(* Logix 5000 project; controller RN21_Architecture 1769-L16ER-BB1B rev 35.11; software revision 35.00; part 9 of 9 *)
(* tags used below, declared in another part *)
   Delformovingupdatedtimertonewpswd : TIMER;
   EmgLoginDn : BOOL;
   ExpDays_NoofattemptsLeft_visb : BOOL;
   ExpDays_NoofattemptsLeft_visbility : BOOL;
   ExpiryDays_MovFrmSrv : DINT;
   FC_RP_Arch : AOI_RP_Arch;
   FCI_PrintInterval : INT;
   FCI_RPDataLogTrig : BOOL;
   HMI_ChangePswd : BOOL;
   HMI_CONTROL_SCREEN : DINT;
   INTERNAL_RN21_HB_PLC2ServerCommFailed : BOOL;
   Lockout_Visb : BOOL;
   Logged_User : STRING;
   MaskTag : STRING;
   MaskTag1 : STRING;
   New_Pswd : STRING;
   New_Pswd_mask : STRING;
   New_Pswd_mask1 : STRING;
   Password_Change_Yes_Button_In_HMI : BOOL;
   PLC_RTC : DINT[7];
   Pswd_UpadatedSuccessfully : BOOL;
   pwdons : BOOL;
   RecipeEntryFloat : REAL[20];
   RecipeEntryInt : INT[11];
   RM_Param1 : DINT;
   RM_Param10 : REAL;
   RM_Param2 : DINT;
   RM_Param3 : DINT;
   RM_Param4 : DINT;
   RM_Param5 : DINT;
   RM_Param6 : REAL;
   RM_Param7 : REAL;
   RM_Param8 : REAL;
   RM_Param9 : REAL;
   RN21_BMAN_HMIBatchStart : BOOL;   // BATCH START
   RN21_LBStatus : INT;   // Login Block Status
   RN21_RM_LOADDLYBIT : BOOL;
   RN21_UM_ActiveUserMovFrmSrv : DINT;
   RN21_UM_Empty : STRING;   // Whenever Logout Will happen moving the Empty
   RN21_UM_ExpiryBitMovFrmSrv : DINT;
   RN21_UM_HMIPSWD_Visb : BOOL;
   RN21_UM_HMIPSWDAPPLY : BOOL;
   RN21_UM_HMIUserIDApply : BOOL;
   RN21_UM_HMIUSERPSWD : STRING;
   RN21_UM_INVALIDUserLatch : BOOL;
   RN21_UM_MaintBit : BOOL;
   RN21_UM_OperBit : BOOL;
   RN21_UM_Status_Visb : BOOL;
   RN21_UM_SupBit : BOOL;
   RN21_UM_USERIDEquLatch : BOOL;
   RN21_UM_USERIDMovFrmSrv : STRING;
   RN21_UM_UserLogout : BOOL;
   RN21_UM_UserLvlMovFrmSrv : DINT;
   RN21_UMAdmBit : BOOL;
   RN21_UMLogoutTag : INT;
   RN21_UMONS : DINT;
   RN21_UserLoginDN : BOOL;
   RP_Param1 : DINT;
   RP_Param10 : REAL;
   RP_Param2 : DINT;
   RP_Param3 : DINT;
   RP_Param4 : DINT;
   RP_Param5 : DINT;
   RP_Param6 : REAL;
   RP_Param7 : REAL;
   RP_Param8 : REAL;
   RP_Param9 : REAL;
   RPSrc : UDT_Recipe;
   RPSrc_RP_UID : DINT;
   TMR_LOGOUT : TIMER;
   TMR_UMLogoutTag : TIMER;
   TMR_UserIDRstDly : TIMER;
   TMRHMIPSWDVisb_Dly : TIMER;
   UM_Status1 : DINT;
   DummyBit : BOOL;
   EmergencyLoginActivated_Bit : BOOL;
   EmergencyUserIDEqual : BOOL;
   EmergencyUserPaswdEqual : BOOL;
   RN21_EmgUserID : STRING;
   RN21_UM_EmgPSWD : STRING;
   RP_Trigger : BOOL;
   RP_UID : DINT;
   RPSer : UDT_Recipe;
   UM_ACT : DINT;
   UM_Confirmation_Bit : BOOL;
   UM_EXPIRY : DINT;
   UM_EXPIRY_DAYS : DINT;
   UM_lockoutDurationLeft : DINT;
   UM_LVL : DINT;
   UM_NoOfAttempts : DINT;
   UM_PWD : STRING;
   UM_Status : DINT;
   UM_UID : STRING;
   UM_UID_OUT : STRING;
   UM_UniqueID : DINT;
(* MainProgram, continued *)

ROUTINE RN21_RM_Map   (* ladder *)
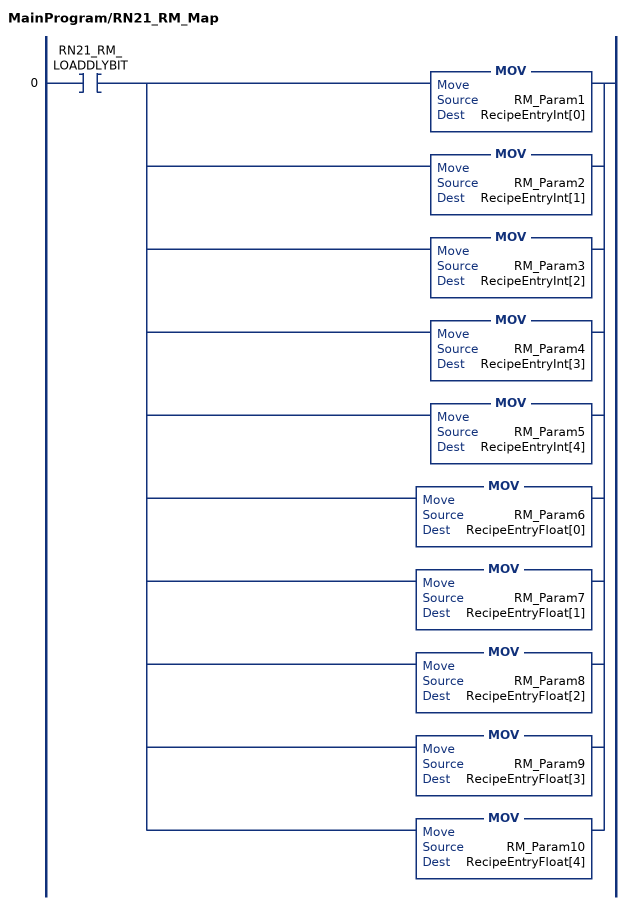
   0: XIC(RN21_RM_LOADDLYBIT)[MOV(RM_Param1,RecipeEntryInt[0]) ,MOV(RM_Param2,RecipeEntryInt[1]) ,MOV(RM_Param3,RecipeEntryInt[2]) ,MOV(RM_Param4,RecipeEntryInt[3]) ,MOV(RM_Param5,RecipeEntryInt[4]) ,MOV(RM_Param6,RecipeEntryFloat[0]) ,MOV(RM_Param7,RecipeEntryFloat[1]) ,MOV(RM_Param8,RecipeEntryFloat[2]) ,MOV(RM_Param9,RecipeEntryFloat[3]) ,MOV(RM_Param10,RecipeEntryFloat[4]) ];
END_ROUTINE

ROUTINE RN21_RP_Main   (* ladder *)
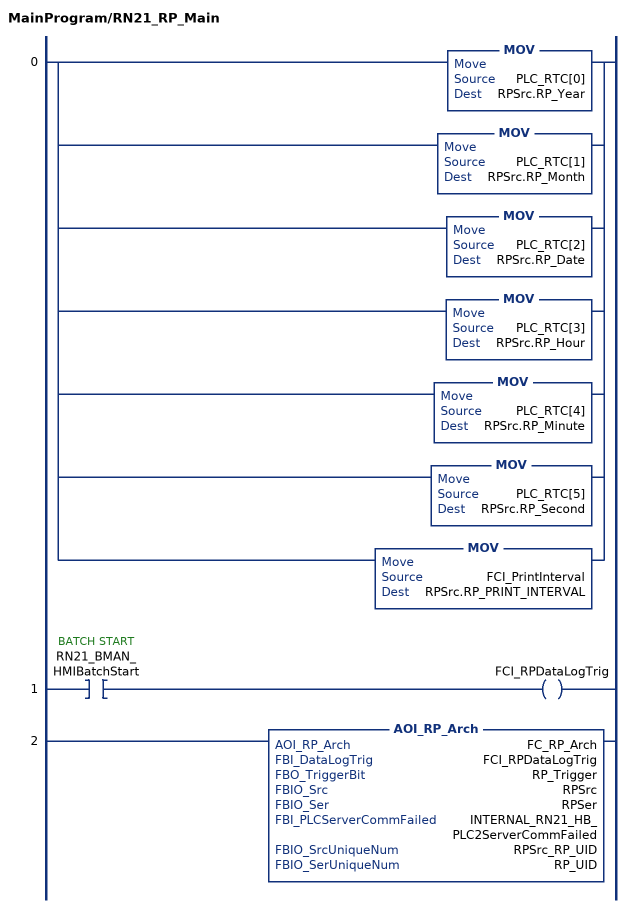
   0: [MOV(PLC_RTC[0],RPSrc.RP_Year) ,MOV(PLC_RTC[1],RPSrc.RP_Month) ,MOV(PLC_RTC[2],RPSrc.RP_Date) ,MOV(PLC_RTC[3],RPSrc.RP_Hour) ,MOV(PLC_RTC[4],RPSrc.RP_Minute) ,MOV(PLC_RTC[5],RPSrc.RP_Second) ,MOV(FCI_PrintInterval,RPSrc.RP_PRINT_INTERVAL) ];
   1: XIC(RN21_BMAN_HMIBatchStart)OTE(FCI_RPDataLogTrig);
   2: AOI_RP_Arch(FC_RP_Arch,FCI_RPDataLogTrig,RP_Trigger,RPSrc,RPSer,INTERNAL_RN21_HB_PLC2ServerCommFailed,RPSrc_RP_UID,RP_UID);
END_ROUTINE

ROUTINE RN21_RP_Map   (* ladder *)
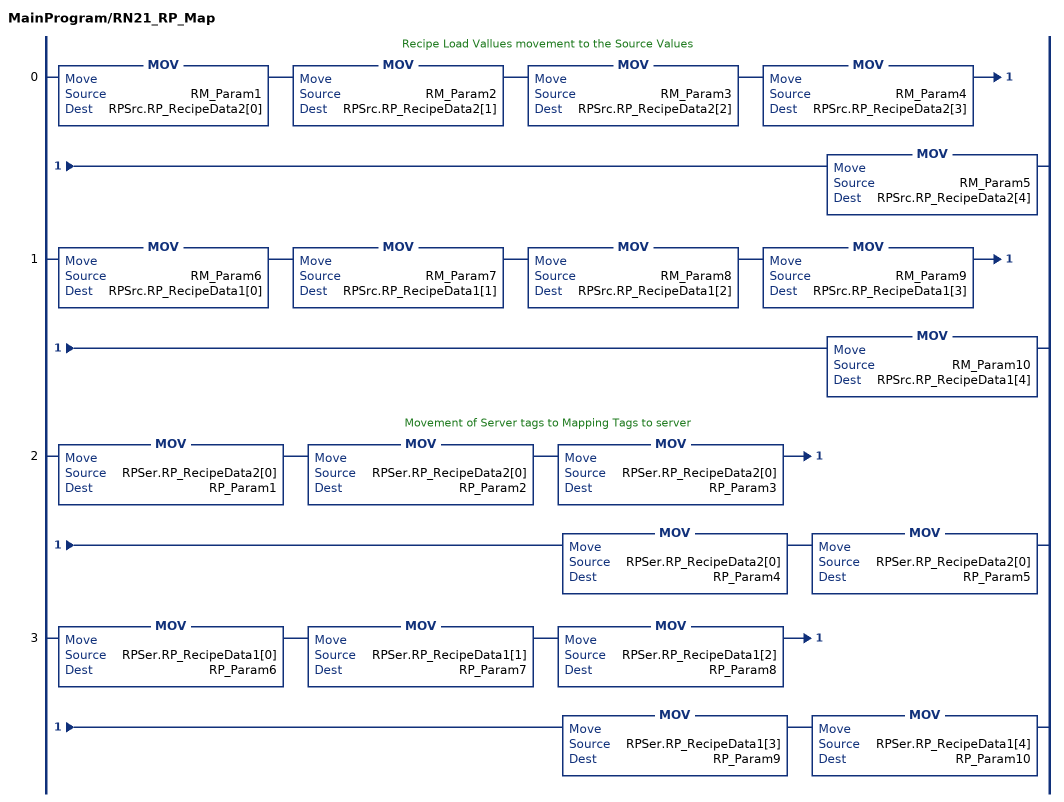
   // Recipe Load Vallues movement to the Source Values
   0: MOV(RM_Param1,RPSrc.RP_RecipeData2[0])MOV(RM_Param2,RPSrc.RP_RecipeData2[1])MOV(RM_Param3,RPSrc.RP_RecipeData2[2])MOV(RM_Param4,RPSrc.RP_RecipeData2[3])MOV(RM_Param5,RPSrc.RP_RecipeData2[4]);
   1: MOV(RM_Param6,RPSrc.RP_RecipeData1[0])MOV(RM_Param7,RPSrc.RP_RecipeData1[1])MOV(RM_Param8,RPSrc.RP_RecipeData1[2])MOV(RM_Param9,RPSrc.RP_RecipeData1[3])MOV(RM_Param10,RPSrc.RP_RecipeData1[4]);
   // Movement of Server tags to Mapping Tags to server
   2: MOV(RPSer.RP_RecipeData2[0],RP_Param1)MOV(RPSer.RP_RecipeData2[0],RP_Param2)MOV(RPSer.RP_RecipeData2[0],RP_Param3)MOV(RPSer.RP_RecipeData2[0],RP_Param4)MOV(RPSer.RP_RecipeData2[0],RP_Param5);
   3: MOV(RPSer.RP_RecipeData1[0],RP_Param6)MOV(RPSer.RP_RecipeData1[1],RP_Param7)MOV(RPSer.RP_RecipeData1[2],RP_Param8)MOV(RPSer.RP_RecipeData1[3],RP_Param9)MOV(RPSer.RP_RecipeData1[4],RP_Param10);
END_ROUTINE

ROUTINE RN21_UM_Main   (* ladder *)
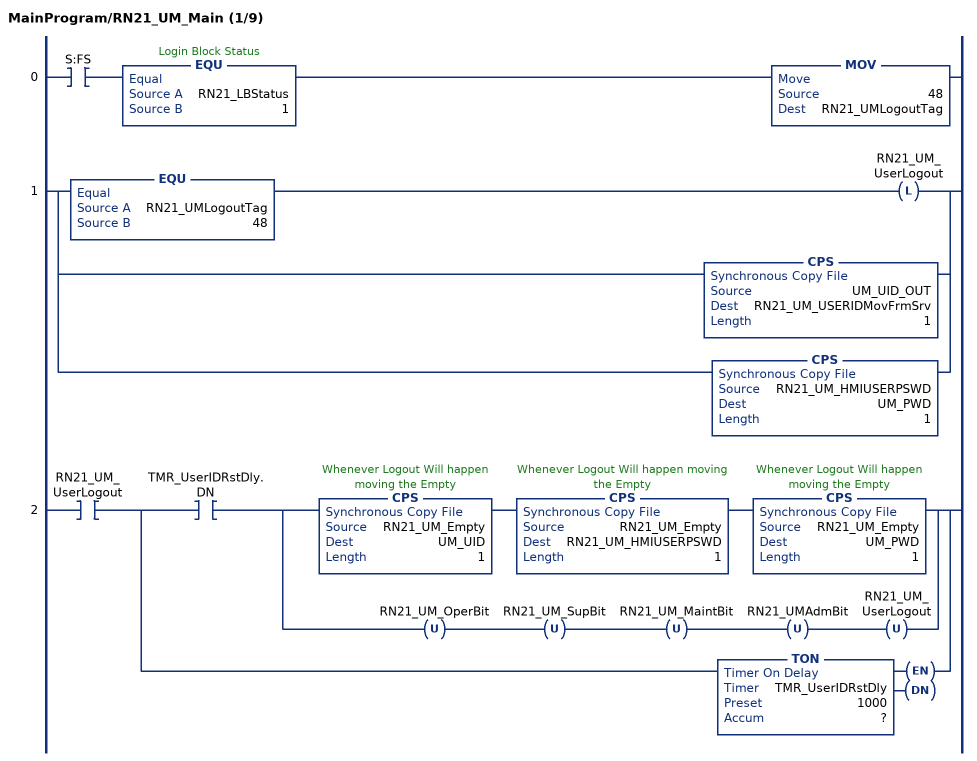
   0: XIC(S:FS)EQU(RN21_LBStatus,1)MOV(48,RN21_UMLogoutTag);
   1: [EQU(RN21_UMLogoutTag,48) OTL(RN21_UM_UserLogout) ,CPS(UM_UID_OUT,RN21_UM_USERIDMovFrmSrv,1) ,CPS(RN21_UM_HMIUSERPSWD,UM_PWD,1) ];
   2: XIC(RN21_UM_UserLogout)[XIC(TMR_UserIDRstDly.DN) [CPS(RN21_UM_Empty,UM_UID,1) CPS(RN21_UM_Empty,RN21_UM_HMIUSERPSWD,1) CPS(RN21_UM_Empty,UM_PWD,1) ,OTU(RN21_UM_OperBit) OTU(RN21_UM_SupBit) OTU(RN21_UM_MaintBit) OTU(RN21_UMAdmBit) OTU(RN21_UM_UserLogout) ] ,TON(TMR_UserIDRstDly,?,?) ];
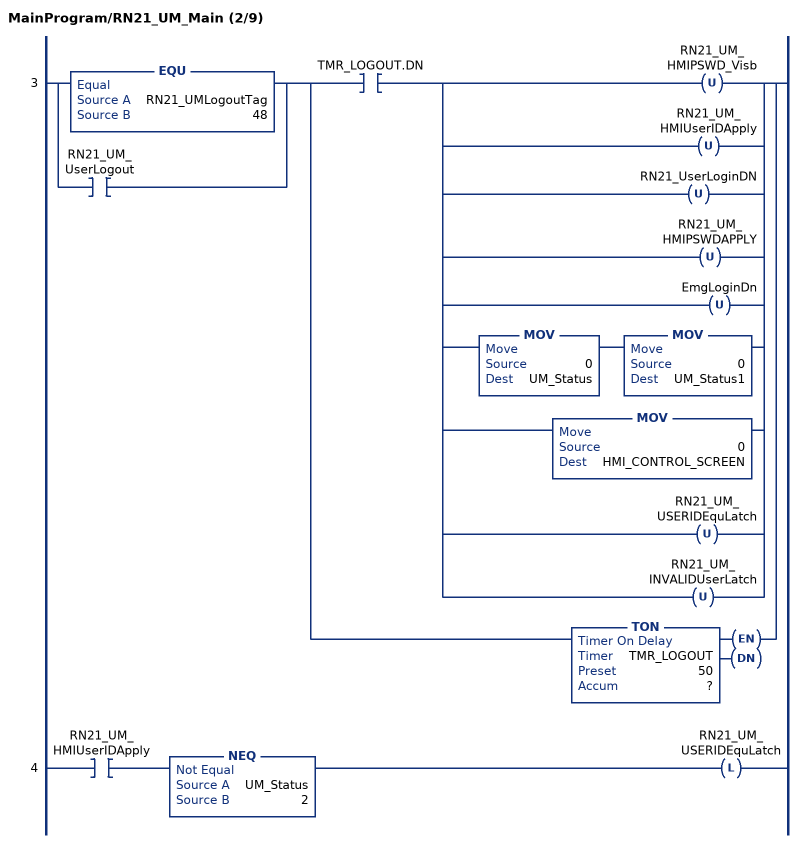
   3: [EQU(RN21_UMLogoutTag,48) ,XIC(RN21_UM_UserLogout) ][XIC(TMR_LOGOUT.DN) [OTU(RN21_UM_HMIPSWD_Visb) ,OTU(RN21_UM_HMIUserIDApply) ,OTU(RN21_UserLoginDN) ,OTU(RN21_UM_HMIPSWDAPPLY) ,OTU(EmgLoginDn) ,MOV(0,UM_Status) MOV(0,UM_Status1) ,MOV(0,HMI_CONTROL_SCREEN) ,OTU(RN21_UM_USERIDEquLatch) ,OTU(RN21_UM_INVALIDUserLatch) ] ,TON(TMR_LOGOUT,?,?) ];
   4: XIC(RN21_UM_HMIUserIDApply)NEQ(UM_Status,2)OTL(RN21_UM_USERIDEquLatch);
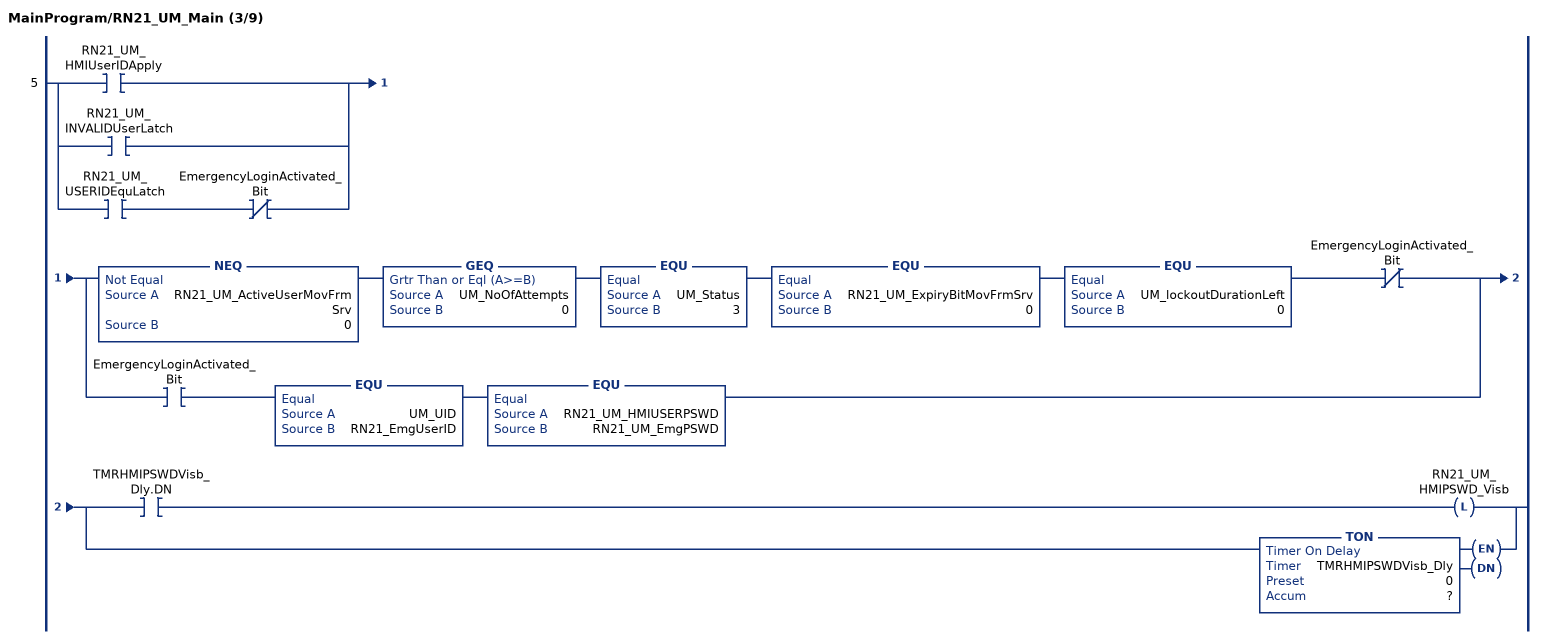
   5: [XIC(RN21_UM_HMIUserIDApply) ,XIC(RN21_UM_INVALIDUserLatch) ,XIC(RN21_UM_USERIDEquLatch) XIO(EmergencyLoginActivated_Bit) ][NEQ(RN21_UM_ActiveUserMovFrmSrv,0) GEQ(UM_NoOfAttempts,0) EQU(UM_Status,3) EQU(RN21_UM_ExpiryBitMovFrmSrv,0) EQU(UM_lockoutDurationLeft,0) XIO(EmergencyLoginActivated_Bit) ,XIC(EmergencyLoginActivated_Bit) EQU(UM_UID,RN21_EmgUserID) EQU(RN21_UM_HMIUSERPSWD,RN21_UM_EmgPSWD) ][XIC(TMRHMIPSWDVisb_Dly.DN) OTL(RN21_UM_HMIPSWD_Visb) ,TON(TMRHMIPSWDVisb_Dly,?,?) ];
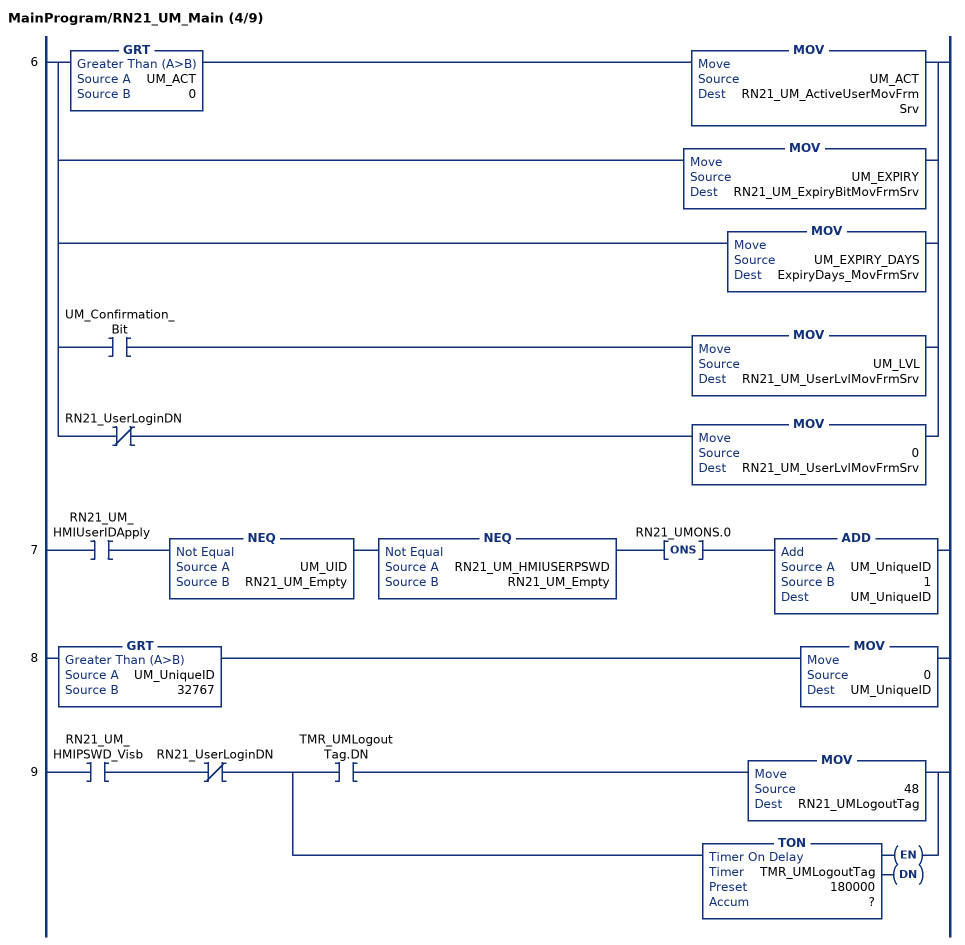
   6: [GRT(UM_ACT,0) MOV(UM_ACT,RN21_UM_ActiveUserMovFrmSrv) ,MOV(UM_EXPIRY,RN21_UM_ExpiryBitMovFrmSrv) ,MOV(UM_EXPIRY_DAYS,ExpiryDays_MovFrmSrv) ,XIC(UM_Confirmation_Bit) MOV(UM_LVL,RN21_UM_UserLvlMovFrmSrv) ,XIO(RN21_UserLoginDN) MOV(0,RN21_UM_UserLvlMovFrmSrv) ];
   7: XIC(RN21_UM_HMIUserIDApply)NEQ(UM_UID,RN21_UM_Empty)NEQ(RN21_UM_HMIUSERPSWD,RN21_UM_Empty)ONS(RN21_UMONS.0)ADD(UM_UniqueID,1,UM_UniqueID);
   8: GRT(UM_UniqueID,32767)MOV(0,UM_UniqueID);
   9: XIC(RN21_UM_HMIPSWD_Visb)XIO(RN21_UserLoginDN)[XIC(TMR_UMLogoutTag.DN) MOV(48,RN21_UMLogoutTag) ,TON(TMR_UMLogoutTag,?,?) ];
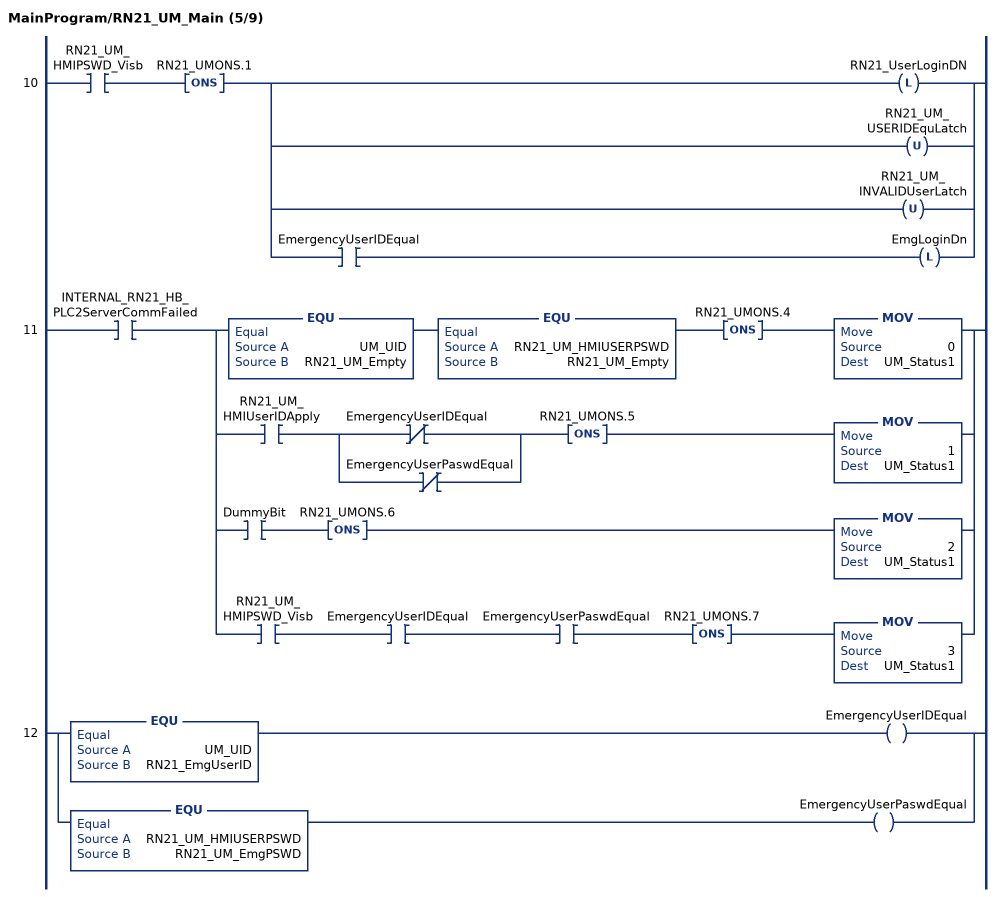
   10: XIC(RN21_UM_HMIPSWD_Visb)ONS(RN21_UMONS.1)[OTL(RN21_UserLoginDN) ,OTU(RN21_UM_USERIDEquLatch) ,OTU(RN21_UM_INVALIDUserLatch) ,XIC(EmergencyUserIDEqual) OTL(EmgLoginDn) ];
   11: XIC(INTERNAL_RN21_HB_PLC2ServerCommFailed)[EQU(UM_UID,RN21_UM_Empty) EQU(RN21_UM_HMIUSERPSWD,RN21_UM_Empty) ONS(RN21_UMONS.4) MOV(0,UM_Status1) ,XIC(RN21_UM_HMIUserIDApply) [XIO(EmergencyUserIDEqual) ,XIO(EmergencyUserPaswdEqual) ] ONS(RN21_UMONS.5) MOV(1,UM_Status1) ,XIC(DummyBit) ONS(RN21_UMONS.6) MOV(2,UM_Status1) ,XIC(RN21_UM_HMIPSWD_Visb) XIC(EmergencyUserIDEqual) XIC(EmergencyUserPaswdEqual) ONS(RN21_UMONS.7) MOV(3,UM_Status1) ];
   12: [EQU(UM_UID,RN21_EmgUserID) OTE(EmergencyUserIDEqual) ,EQU(RN21_UM_HMIUSERPSWD,RN21_UM_EmgPSWD) OTE(EmergencyUserPaswdEqual) ];
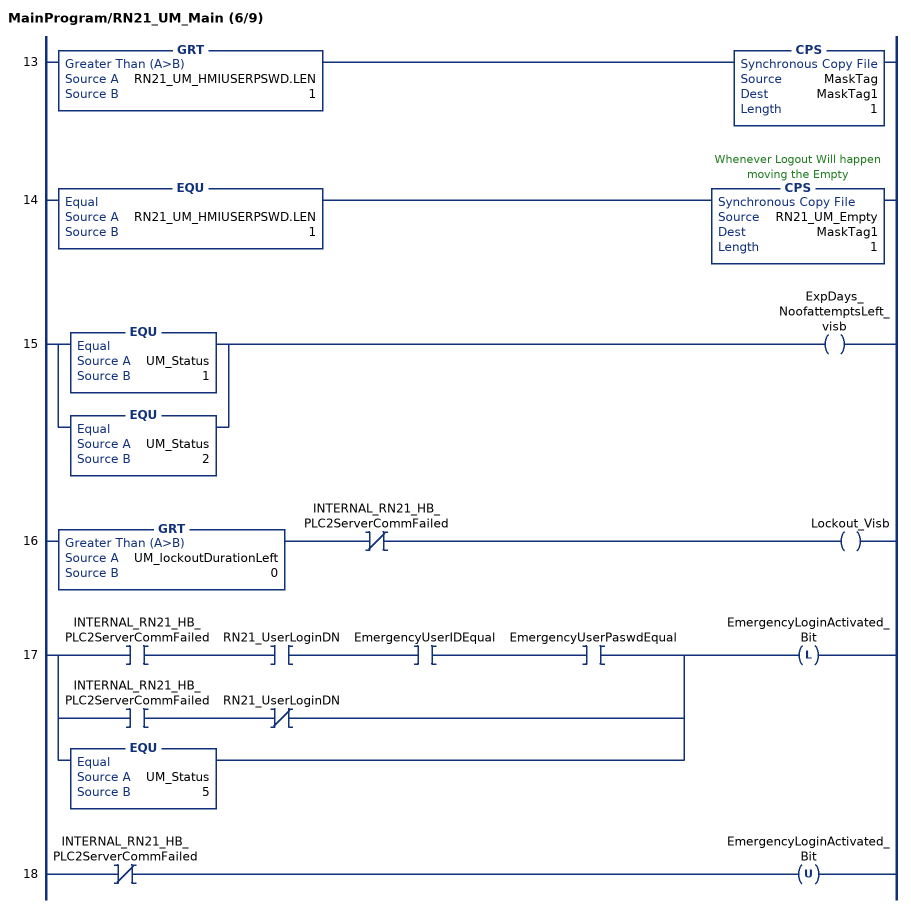
   13: GRT(RN21_UM_HMIUSERPSWD.LEN,1)CPS(MaskTag,MaskTag1,1);
   14: EQU(RN21_UM_HMIUSERPSWD.LEN,1)CPS(RN21_UM_Empty,MaskTag1,1);
   15: [EQU(UM_Status,1) ,EQU(UM_Status,2) ]OTE(ExpDays_NoofattemptsLeft_visb);
   16: GRT(UM_lockoutDurationLeft,0)XIO(INTERNAL_RN21_HB_PLC2ServerCommFailed)OTE(Lockout_Visb);
   17: [XIC(INTERNAL_RN21_HB_PLC2ServerCommFailed) XIC(RN21_UserLoginDN) XIC(EmergencyUserIDEqual) XIC(EmergencyUserPaswdEqual) ,XIC(INTERNAL_RN21_HB_PLC2ServerCommFailed) XIO(RN21_UserLoginDN) ,EQU(UM_Status,5) ]OTL(EmergencyLoginActivated_Bit);
   18: XIO(INTERNAL_RN21_HB_PLC2ServerCommFailed)OTU(EmergencyLoginActivated_Bit);
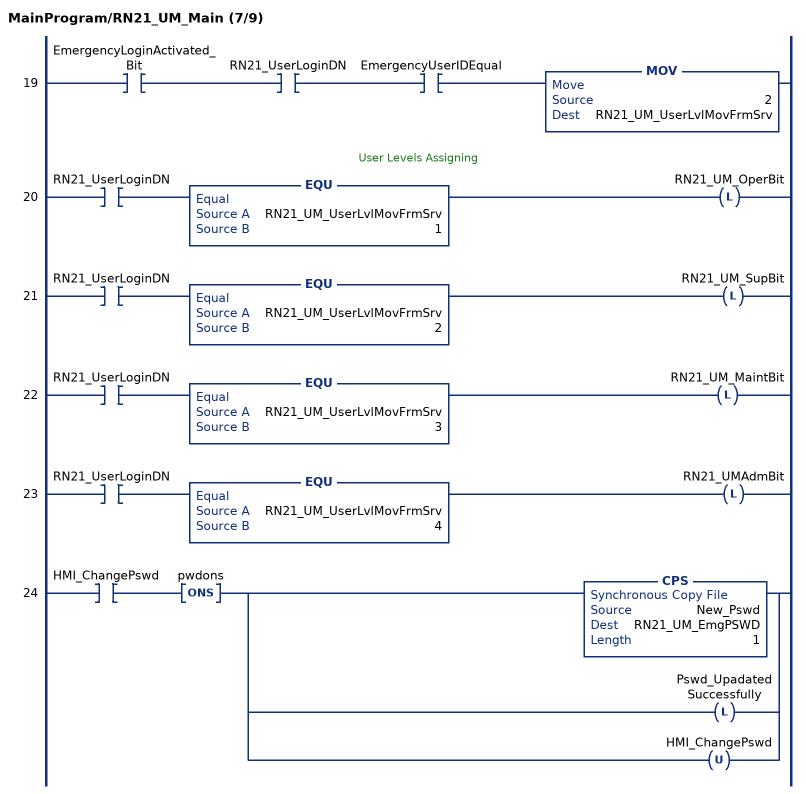
   19: XIC(EmergencyLoginActivated_Bit)XIC(RN21_UserLoginDN)XIC(EmergencyUserIDEqual)MOV(2,RN21_UM_UserLvlMovFrmSrv);
   // User Levels Assigning
   20: XIC(RN21_UserLoginDN)EQU(RN21_UM_UserLvlMovFrmSrv,1)OTL(RN21_UM_OperBit);
   21: XIC(RN21_UserLoginDN)EQU(RN21_UM_UserLvlMovFrmSrv,2)OTL(RN21_UM_SupBit);
   22: XIC(RN21_UserLoginDN)EQU(RN21_UM_UserLvlMovFrmSrv,3)OTL(RN21_UM_MaintBit);
   23: XIC(RN21_UserLoginDN)EQU(RN21_UM_UserLvlMovFrmSrv,4)OTL(RN21_UMAdmBit);
   24: XIC(HMI_ChangePswd)ONS(pwdons)[CPS(New_Pswd,RN21_UM_EmgPSWD,1) ,OTL(Pswd_UpadatedSuccessfully) ,OTU(HMI_ChangePswd) ];
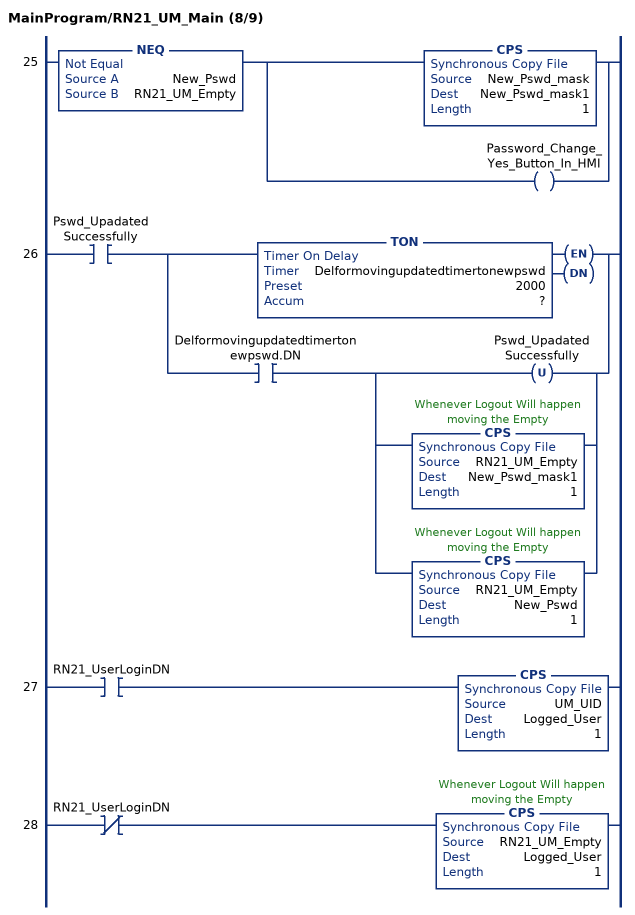
   25: NEQ(New_Pswd,RN21_UM_Empty)[CPS(New_Pswd_mask,New_Pswd_mask1,1) ,OTE(Password_Change_Yes_Button_In_HMI) ];
   26: XIC(Pswd_UpadatedSuccessfully)[TON(Delformovingupdatedtimertonewpswd,?,?) ,XIC(Delformovingupdatedtimertonewpswd.DN) [OTU(Pswd_UpadatedSuccessfully) ,CPS(RN21_UM_Empty,New_Pswd_mask1,1) ,CPS(RN21_UM_Empty,New_Pswd,1) ] ];
   27: XIC(RN21_UserLoginDN)CPS(UM_UID,Logged_User,1);
   28: XIO(RN21_UserLoginDN)CPS(RN21_UM_Empty,Logged_User,1);
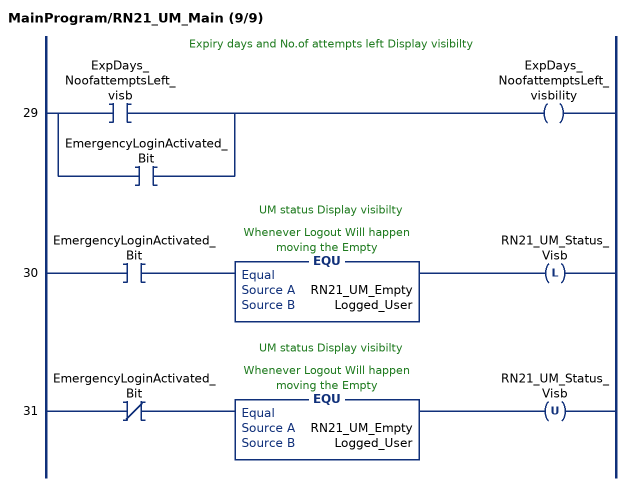
   // Expiry days and No.of attempts left Display visibilty
   29: [XIC(ExpDays_NoofattemptsLeft_visb) ,XIC(EmergencyLoginActivated_Bit) ]OTE(ExpDays_NoofattemptsLeft_visbility);
   // UM status Display visibilty
   30: XIC(EmergencyLoginActivated_Bit)EQU(RN21_UM_Empty,Logged_User)OTL(RN21_UM_Status_Visb);
   // UM status Display visibilty
   31: XIO(EmergencyLoginActivated_Bit)EQU(RN21_UM_Empty,Logged_User)OTU(RN21_UM_Status_Visb);
END_ROUTINE
END_PROGRAM
